FUNCTION_BLOCK FB_Test_1
VAR_INPUT
	ins_CommIn			:Type_CommIn_Test;
	inint_Position		:INT;
	inm_Reset			:BOOL;
	inlreal_RandomNumber:LREAL;
END_VAR
VAR_OUTPUT
	outs_CommOut		:Type_CommOut_Test;
	outm_StartTimer		:BOOL;
	o_AverageCycleTime  :REAL;

END_VAR
VAR
	time_TimerInput		:TIME;
	FB_RAND				:DRAND;
	m_Stop				:BOOL;
	m_First				:BOOL;
	m_FirstCycleTime	:BOOL;
	
	o_TotalCycleTime	:BYTE;
	o_PartExists		:BOOL;
	
	RetVal 				:enum_RetVal;
	
	o_ProcessCycleTime	:BYTE;
	(*	Timers	*)
	lreal_TimerInput			:LREAL;
	T03_Check_Holes				:TON;
	T04_Check_Dust				:TON;
	T05_Check_Sharp_Edges		:TON;
	
	Instance_CountTotalCycleTime		:FB_CountCycleTime();
	Instance_CountProcessCycleTime		:FB_CountCycleTime();

	
	time_Timer_RandomInput: TIME;
END_VAR

IF inm_Reset = FALSE
	THEN
	SFCReset:=FALSE;
	A01_AutomaticMode();
	
	ELSE
		SFCReset:=TRUE;
		A01_AutomaticMode();
END_IF

ACTION A01_AutomaticMode:
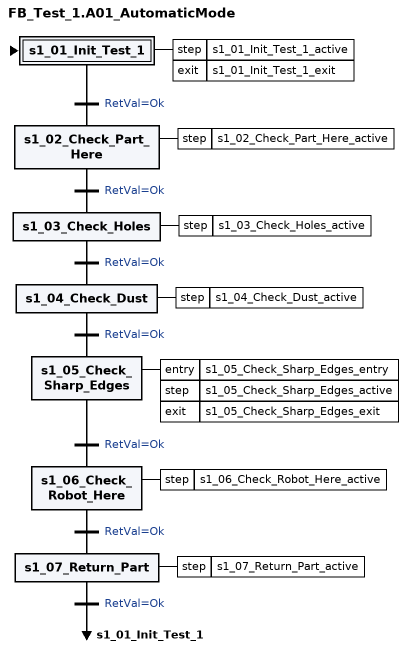
INITIAL_STEP s1_01_Init_Test_1:
    s1_01_Init_Test_1_active(N);  // step action
    s1_01_Init_Test_1_exit(P0);  // exit action
END_STEP
TRANSITION FROM s1_01_Init_Test_1 TO s1_02_Check_Part_Here
    := RetVal=Ok;
END_TRANSITION
STEP s1_02_Check_Part_Here:
    s1_02_Check_Part_Here_active(N);  // step action
END_STEP
TRANSITION FROM s1_02_Check_Part_Here TO s1_03_Check_Holes
    := RetVal=Ok;
END_TRANSITION
STEP s1_03_Check_Holes:
    s1_03_Check_Holes_active(N);  // step action
END_STEP
TRANSITION FROM s1_03_Check_Holes TO s1_04_Check_Dust
    := RetVal=Ok;
END_TRANSITION
STEP s1_04_Check_Dust:
    s1_04_Check_Dust_active(N);  // step action
END_STEP
TRANSITION FROM s1_04_Check_Dust TO s1_05_Check_Sharp_Edges
    := RetVal=Ok;
END_TRANSITION
STEP s1_05_Check_Sharp_Edges:
    s1_05_Check_Sharp_Edges_entry(P1);  // entry action
    s1_05_Check_Sharp_Edges_active(N);  // step action
    s1_05_Check_Sharp_Edges_exit(P0);  // exit action
END_STEP
TRANSITION FROM s1_05_Check_Sharp_Edges TO s1_06_Check_Robot_Here
    := RetVal=Ok;
END_TRANSITION
STEP s1_06_Check_Robot_Here:
    s1_06_Check_Robot_Here_active(N);  // step action
END_STEP
TRANSITION FROM s1_06_Check_Robot_Here TO s1_07_Return_Part
    := RetVal=Ok;
END_TRANSITION
STEP s1_07_Return_Part:
    s1_07_Return_Part_active(N);  // step action
END_STEP
TRANSITION FROM s1_07_Return_Part TO s1_01_Init_Test_1
    := RetVal=Ok;
END_TRANSITION
END_ACTION

ACTION s1_01_Init_Test_1_active:
RetVal:=Running;

Instance_CountTotalCycleTime(inm_TimeActive:=FALSE);
o_TotalCycleTime:=REAL_TO_BYTE(Instance_CountTotalCycleTime.outr_CycleTime);

outs_CommOut.s_Robot.m_Empty:=TRUE;
outs_CommOut.s_Robot.m_Ready:=FALSE;

IF  ins_CommIn.s_Robot.m_OutOfArea
	THEN
	Instance_CountTotalCycleTime(inm_TimeActive:=TRUE);	
	RetVal:=Ok;
END_IF
END_ACTION

ACTION s1_01_Init_Test_1_exit:
IF NOT m_FirstCycleTime
	THEN
	o_AverageCycleTime := 105;
END_IF
END_ACTION

ACTION s1_02_Check_Part_Here_active:
RetVal:=Running;

IF ins_CommIn.s_Robot.m_OutOfArea = FALSE
	AND ins_CommIn.s_Robot.m_Work = FALSE
	THEN
	outs_CommOut.s_Robot.m_Empty:=FALSE;
END_IF

IF ins_CommIn.s_Robot.m_PartDropped
	THEN
	Instance_CountProcessCycleTime(inm_TimeActive:=TRUE);
	RetVal:=Ok;
END_IF
END_ACTION

ACTION s1_03_Check_Holes_active:
RetVal:=Running;

T03_Check_Holes(IN:=TRUE,PT:=T#5s);

IF T03_Check_Holes.Q
	THEN
	T03_Check_Holes(IN:=FALSE);
	RetVal:=Ok;
END_IF
END_ACTION

ACTION s1_04_Check_Dust_active:
RetVal:=Running;

T04_Check_Dust(IN:=TRUE,PT:=T#5S);

IF T04_Check_Dust.Q
	THEN
	T04_Check_Dust(IN:=FALSE);
	RetVal:=Ok;
END_IF
END_ACTION

ACTION s1_05_Check_Sharp_Edges_active:
RetVal:=Running;

time_TimerInput:=LREAL_TO_TIME(lreal_TimerInput*100000);

T05_Check_Sharp_Edges(IN:=TRUE,PT:=T#95S);
		
IF T05_Check_Sharp_Edges.Q
	THEN	
	Instance_CountProcessCycleTime(inm_TimeActive:=FALSE);
	o_ProcessCycleTime:=REAL_TO_BYTE(Instance_CountProcessCycleTime.outr_CycleTime);
	
	IF m_First 
	THEN
		o_AverageCycleTime:= (o_AverageCycleTime + o_ProcessCycleTime)/2;
		ELSE
		o_AverageCycleTime := o_ProcessCycleTime;
	END_IF
	
	outs_CommOut.s_Robot.m_Ready:=TRUE;
	o_PartExists:=TRUE;
	
	ADSLOGSTR(msgCtrlMask:= ADSLOG_MSGTYPE_WARN,
		msgFmtStr:='The time is: %s ms ',
		strArg:=LREAL_TO_STRING(lreal_TimerInput*100000));
	
	T05_Check_Sharp_Edges(IN:=FALSE);
	m_Stop:=FALSE;
	RetVal:=Ok;
END_IF
END_ACTION

ACTION s1_05_Check_Sharp_Edges_entry:
lreal_TimerInput:=inlreal_RandomNumber;
END_ACTION

ACTION s1_05_Check_Sharp_Edges_exit:
m_First:=TRUE;
END_ACTION

ACTION s1_06_Check_Robot_Here_active:
RetVal:=Running;

IF ins_CommIn.s_Robot.m_OutOfArea = FALSE
	THEN
	RetVal:=Ok;
END_IF
END_ACTION

ACTION s1_07_Return_Part_active:
RetVal:=Running;
m_FirstCycleTime:=TRUE;
o_PartExists:=FALSE;

IF ins_CommIn.s_Robot.m_Work = FALSE
	AND ins_CommIn.s_Robot.m_PartDropped = FALSE
	THEN
	RetVal:=Ok;
END_IF
END_ACTION

END_FUNCTION_BLOCK

(* stored: Version 1.1.0.1, ProductVersion 3.1.4024.3
   POU FB_Test_1: Id {b9ae1877-fe24-4421-862b-04e2e0499a4b}, SpecialFunc None
   Folder S1: Id {9e7f4295-f43e-416b-90e2-0afa9d1256c8}
   Folder S2: Id {40c39097-a828-483a-a7c5-acb7748b72bd}
   Action A01_AutomaticMode: Id {9e8f7977-6b36-45a2-851c-40f9f604888e}
   Action s1_01_Init_Test_1_active: Id {9253b2ef-ab28-4995-957a-6139ae70938b}
   Action s1_01_Init_Test_1_exit: Id {3aadb0cd-c354-46fc-a327-943cfbb8b4e7}
   Action s1_02_Check_Part_Here_active: Id {4508e249-55d1-4fe9-83a2-08944b9fd2bf}
   Action s1_03_Check_Holes_active: Id {4f126280-faa2-4630-b982-36b38ab81b0e}
   Action s1_04_Check_Dust_active: Id {3227dc78-aafc-4327-aee6-3acc3e353e50}
   Action s1_05_Check_Sharp_Edges_active: Id {88c7d0dc-81b7-4dcf-89b8-07e6f8c6c28d}
   Action s1_05_Check_Sharp_Edges_entry: Id {46731ec6-60bd-4fae-a9b3-3a568e5bc974}
   Action s1_05_Check_Sharp_Edges_exit: Id {bdb03688-4e57-440b-909a-1a0ee32f80ee}
   Action s1_06_Check_Robot_Here_active: Id {2777cd57-218f-4831-ab8d-14f87fb238e6}
   Action s1_07_Return_Part_active: Id {81d5f8ee-0be0-429a-afb0-6a056400a1e4} *)
